Staubli VAL3: OnF6.pgx

program OnF6()
begin
end
